KUKA KRL data list: PulsGen12ms.dat

&ACCESS RV1
DEFDAT PulsGen12ms PUBLIC

ENDDAT
